(* PLC project car, Dassault Systèmes ControlBuild 2024x *)
(* stored: creationDateTime 2023-10-03T11:13:52-01:00 *)

PROGRAM tni_train.car
  VAR_INPUT
    AuthorizationClosingLeftC1 : BOOL := false;
    AuthorizationOpeningRightC1 : BOOL := false;
    AuthorizationClosingRightC1 : BOOL := false;
    AuthorizationOpeningLeftC1 : BOOL := false;
  END_VAR
  VAR_INPUT
    AuthorizationClosingLeftC2 : BOOL := false;
    AuthorizationOpeningRightC2 : BOOL := false;
    AuthorizationClosingRightC2 : BOOL := false;
    AuthorizationOpeningLeftC2 : BOOL := false;
  END_VAR
  VAR_OUTPUT
    doorL1Closed : BOOL := false;
    doorL1Opened : BOOL := false;
    doorL1Fault : DINT := 0;
  END_VAR
  VAR_OUTPUT
    doorL2Closed : BOOL := false;
    doorL2Opened : BOOL := false;
    doorL2Fault : DINT := 0;
  END_VAR
  VAR_OUTPUT
    doorL3Closed : BOOL := false;
    doorL3Opened : BOOL := false;
    doorL3Fault : DINT := 0;
  END_VAR
  VAR_OUTPUT
    doorR1Closed : BOOL := false;
    doorR1Opened : BOOL := false;
    doorR1Fault : DINT := 0;
  END_VAR
  VAR_OUTPUT
    doorR2Closed : BOOL := false;
    doorR2Opened : BOOL := false;
    doorR2Fault : DINT := 0;
  END_VAR
  VAR_OUTPUT
    doorR3Closed : BOOL := false;
    doorR3Opened : BOOL := false;
    doorR3Fault : DINT := 0;
  END_VAR
  VAR_OUTPUT
    AlarmD1L : BOOL := false;
    AlarmD2L : BOOL := false;
    AlarmD3L : BOOL := false;
    AlarmD1R : BOOL := false;
    AlarmD2R : BOOL := false;
    AlarmD3R : BOOL := false;
  END_VAR

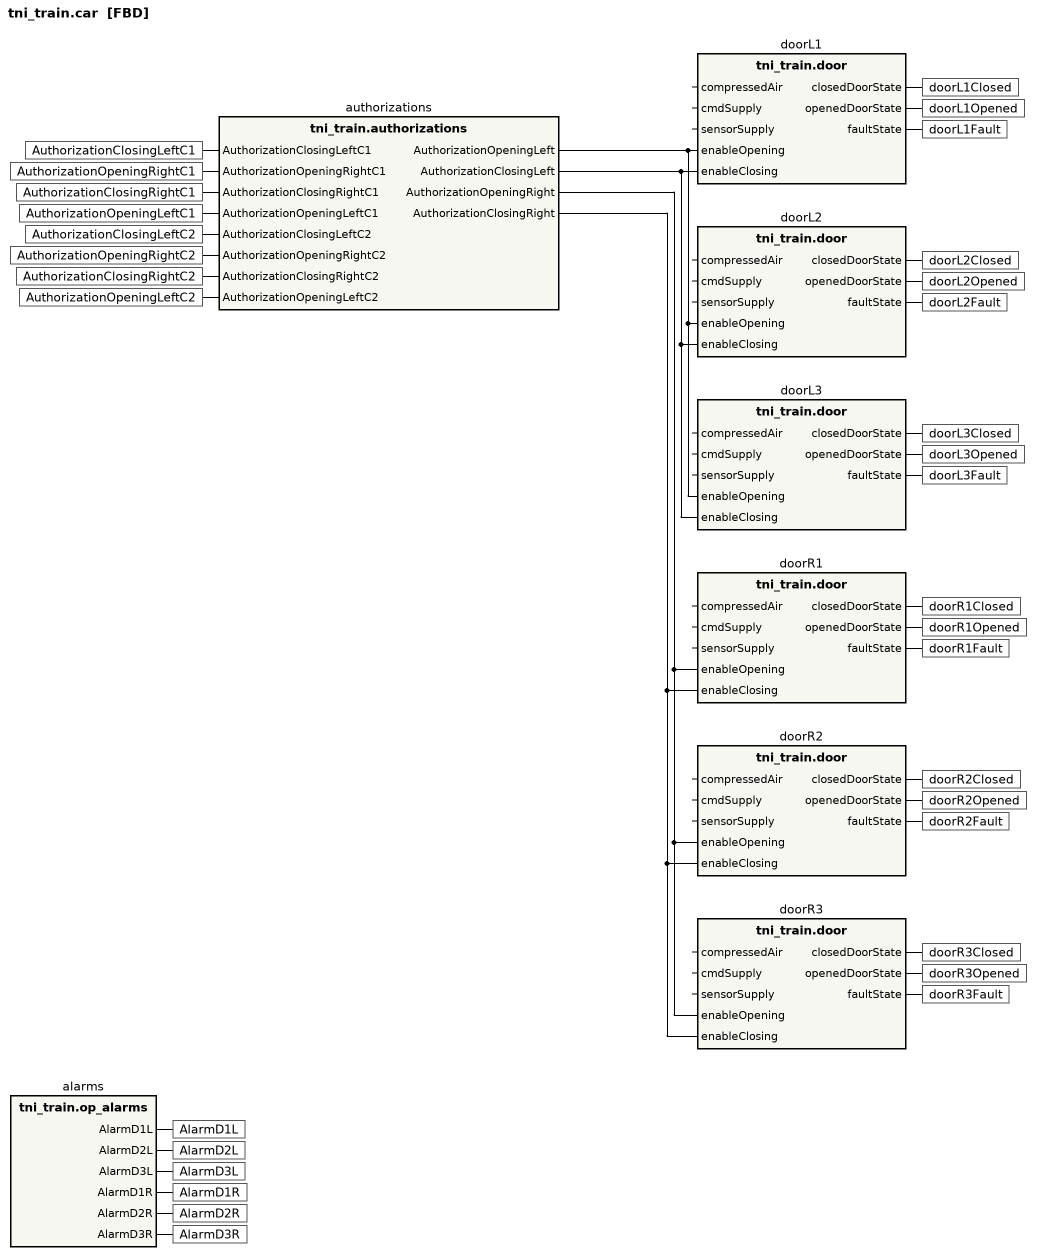
(* FBD diagram, written out as Structured Text *)
authorizations(AuthorizationClosingLeftC1 := AuthorizationClosingLeftC1, AuthorizationOpeningRightC1 := AuthorizationOpeningRightC1, AuthorizationClosingRightC1 := AuthorizationClosingRightC1, AuthorizationOpeningLeftC1 := AuthorizationOpeningLeftC1, AuthorizationClosingLeftC2 := AuthorizationClosingLeftC2, AuthorizationOpeningRightC2 := AuthorizationOpeningRightC2, AuthorizationClosingRightC2 := AuthorizationClosingRightC2, AuthorizationOpeningLeftC2 := AuthorizationOpeningLeftC2);
doorL1(enableOpening := authorizations.AuthorizationOpeningLeft, enableClosing := authorizations.AuthorizationClosingLeft);
doorL1Closed := doorL1.closedDoorState;
doorL1Opened := doorL1.openedDoorState;
doorL1Fault := doorL1.faultState;
doorL2(enableOpening := authorizations.AuthorizationOpeningLeft, enableClosing := authorizations.AuthorizationClosingLeft);
doorL2Closed := doorL2.closedDoorState;
doorL2Opened := doorL2.openedDoorState;
doorL2Fault := doorL2.faultState;
doorL3(enableOpening := authorizations.AuthorizationOpeningLeft, enableClosing := authorizations.AuthorizationClosingLeft);
doorL3Closed := doorL3.closedDoorState;
doorL3Opened := doorL3.openedDoorState;
doorL3Fault := doorL3.faultState;
doorR1(enableOpening := authorizations.AuthorizationOpeningRight, enableClosing := authorizations.AuthorizationClosingRight);
doorR1Closed := doorR1.closedDoorState;
doorR1Opened := doorR1.openedDoorState;
doorR1Fault := doorR1.faultState;
doorR2(enableOpening := authorizations.AuthorizationOpeningRight, enableClosing := authorizations.AuthorizationClosingRight);
doorR2Closed := doorR2.closedDoorState;
doorR2Opened := doorR2.openedDoorState;
doorR2Fault := doorR2.faultState;
alarms();
AlarmD1L := alarms.AlarmD1L;
AlarmD2L := alarms.AlarmD2L;
AlarmD3L := alarms.AlarmD3L;
AlarmD1R := alarms.AlarmD1R;
AlarmD2R := alarms.AlarmD2R;
AlarmD3R := alarms.AlarmD3R;
doorR3(enableOpening := authorizations.AuthorizationOpeningRight, enableClosing := authorizations.AuthorizationClosingRight);
doorR3Closed := doorR3.closedDoorState;
doorR3Opened := doorR3.openedDoorState;
doorR3Fault := doorR3.faultState;
END_PROGRAM
